KUKA KRL program: do_stop2.src

&ACCESS RVO
&REL 15
&PARAM TEMPLATE = C:\KRC\Roboter\Template\FunctionVorgabe
&PARAM EDITMASK = *
def do_stop2()

$fri_to_bool[8] = true
$msg_t.key[] = "stop2 requested                         "
$msg_t.valid = true
brake
$msg_t.key[] = "waiting for fri_bool[8] to resume       "
$msg_t.valid = true
wait for $fri_frm_bool[8] == false

end
